PROGRAM prgMain
VAR
	m_Command_Knetzgau_RESET					: BOOL;							//{#lynus.ag#()}
	m_out1								AT%Q* 	: BOOL;
	m_In1								AT%I* 	: BOOL;
	m_In2								AT%I* 	: BOOL;
	m_Input_Beacon_Knetzgau						: BOOL;							//{#lynus.ag#()}
	m_Input_Siren_Knetzgau						: BOOL;							//{#lynus.ag#()}
	r_tigt_Start_Reset: R_trig;
	tof_Reset: Tof;
	m_LiveBit_5min_Knetzgau						: BOOL;							//{#lynus.ag#()}
	ton_5Min: Ton;
END_VAR

r_tigt_Start_Reset( CLK := m_Command_Knetzgau_RESET);

tof_Reset(	IN:= r_tigt_Start_Reset.Q, 
			PT:= T#2S , 
			Q=> m_out1, 
			ET=> );

 m_Input_Beacon_Knetzgau		:= 			m_In1;
 m_Input_Siren_Knetzgau			:= 			m_In2;		// nicht ausgeführt
 
  ton_5Min(	In := NOT ton_5min.Q	,
	 		PT := T#5M);
			
IF ton_5min.Q AND m_LiveBit_5min_Knetzgau THEN
	m_LiveBit_5min_Knetzgau := FALSE;
ELSIF  ton_5min.Q AND NOT m_LiveBit_5min_Knetzgau THEN
	m_LiveBit_5min_Knetzgau := TRUE;
END_IF

END_PROGRAM

(* stored: Version 1.1.0.1, ProductVersion 3.1.4024.12
   POU prgMain: Id {03f43f79-b52a-4c77-9c92-6164c90e71c1}, SpecialFunc None *)
